FUNCTION_BLOCK IO_WRITER
  (* Version 1.0, 2005-07-04, Goran Cengic, Chalmers *)
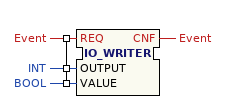
  EVENT_INPUT
    REQ WITH OUTPUT, VALUE;
  END_EVENT
  EVENT_OUTPUT
    CNF;
  END_EVENT
  VAR_INPUT
    OUTPUT : INT; (* The number of the input pin to read from the digital I/O card. *)
    VALUE : BOOL; (* The value to write to the digital I/O card. *)
  END_VAR
END_FUNCTION_BLOCK
